# EPICS autosave request: mw100App/Db/MW100_ADC_slot1_settings.req
$(P)$(DAU):001:Label
$(P)$(DAU):002:Label
$(P)$(DAU):003:Label
$(P)$(DAU):004:Label
$(P)$(DAU):005:Label
$(P)$(DAU):006:Label
$(P)$(DAU):007:Label
$(P)$(DAU):008:Label
$(P)$(DAU):009:Label
$(P)$(DAU):010:Label
